(* PLC project Unnamed, Unknown Unnamed 1 *)
(* stored: creationDateTime 2024-05-18T19:24:04, modificationDateTime 2024-05-18T19:36:35 *)

PROGRAM XOR_and_XNOR
  VAR
    INPUT_0 : BOOL;
    INPUT_1 : BOOL;
    INPUT_2 : BOOL;
    INPUT_3 : BOOL;
    OUTPUT_0 : BOOL;
    OUTPUT_1 : BOOL;
  END_VAR

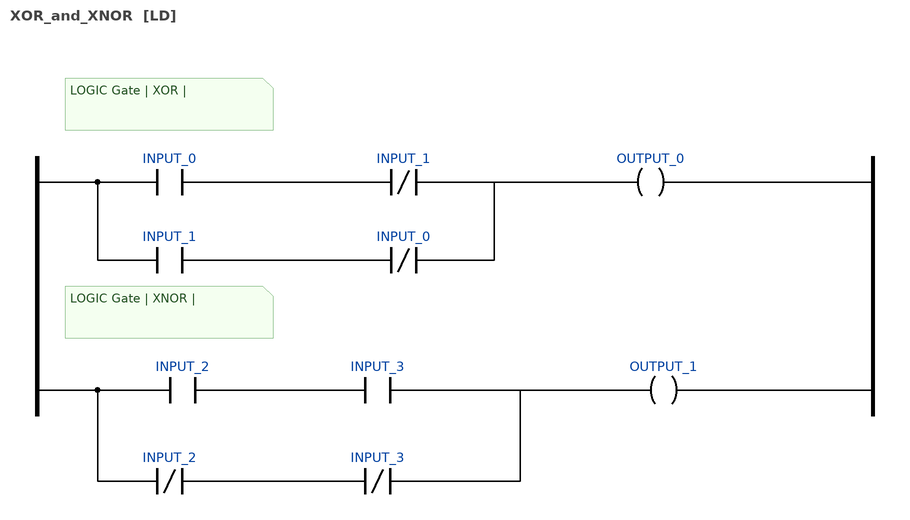
(* LD diagram, written out as Structured Text *)
(* LOGIC Gate | XOR | *)
OUTPUT_0 := INPUT_0 AND NOT INPUT_1 OR INPUT_1 AND NOT INPUT_0;
(* LOGIC Gate | XNOR | *)
OUTPUT_1 := INPUT_2 AND INPUT_3 OR NOT INPUT_2 AND NOT INPUT_3;
END_PROGRAM

CONFIGURATION Config0
  RESOURCE Res0 ON PLC
    TASK task0(INTERVAL := T#20ms, PRIORITY := 0);
    PROGRAM instance0 WITH task0 : XOR_and_XNOR;
  END_RESOURCE
END_CONFIGURATION
